PROGRAM P_ControlBox
VAR
	fbControlBox : FB_ControlBox;
END_VAR

fbControlBox(bRealControlBox := FALSE); // Run controlbox FB with argument. If bRealControlBox is TRUE, then the FB_RealControlBox will be selected when running the program.

END_PROGRAM

(* stored: Version 1.1.0.1, ProductVersion 3.1.4024.12
   POU P_ControlBox: Id {d4f0e33f-2ee9-4ad3-b670-f117d817b486}, SpecialFunc None *)
